// TIA Portal V17 export
// export: Created 2022-03-18T11:15:14.7636384Z, ExportSetting WithDefaults, DisplayName Totally Integrated Automation Portal, DisplayVersion V17, DisplayName TIA Portal Openness, DisplayVersion V17, DisplayName TIA Portal Version Control Interface, DisplayVersion V17, DisplayName SINAMICS Startdrive Advanced, DisplayVersion V17, DisplayName SINAMICS Startdrive G130, G150, S120, S150, SINAMICS MV, S210, DisplayVersion V17, DisplayName SINAMICS Startdrive G110M, G120, G120C, G120D, G120P, G115D, DisplayVersion V17, DisplayName STEP 7 Professional, DisplayVersion V17, DisplayName STEP 7 Safety, DisplayVersion V17, DisplayName WinCC Advanced / Unified PC, DisplayVersion V17
VAR_GLOBAL   // PLC tag table "Default tag table"
   M1_out AT %Q200.0 : "M_out";
   M1_in AT %I200.0 : "M_in";
   M2_out AT %Q219.0 : "M_out";
   M2_in AT %I209.0 : "M_in";
   M3_out AT %Q238.0 : "M_out";
   M3_in AT %I218.0 : "M_in";
   M4_out AT %Q257.0 : "M_out";
   M4_in AT %I227.0 : "M_in";
   M5_out AT %Q276.0 : "M_out";
   M5_in AT %I236.0 : "M_in";
   M6_out AT %Q295.0 : "M_out";
   M6_in AT %I245.0 : "M_in";
   M7_out AT %Q314.0 : "M_out";
   M7_in AT %I254.0 : "M_in";
   M8_out AT %Q333.0 : "M_out";
   M8_in AT %I263.0 : "M_in";
   M9_out AT %Q352.0 : "M_out";
   M9_in AT %I272.0 : "M_in";
   M10_out AT %Q371.0 : "M_out";
   M10_in AT %I281.0 : "M_in";
   M11_out AT %Q390.0 : "M_out";
   M11_in AT %I290.0 : "M_in";
   M12_out AT %Q409.0 : "M_out";
   M12_in AT %I299.0 : "M_in";
   M13_out AT %Q428.0 : "M_out";
   M13_in AT %I308.0 : "M_in";
   M14_out AT %Q447.0 : "M_out";
   M14_in AT %I317.0 : "M_in";
   M15_out AT %Q466.0 : "M_out";
   M15_in AT %I326.0 : "M_in";
   M16_out AT %Q485.0 : "M_out";
   M16_in AT %I335.0 : "M_in";
   M17_out AT %Q504.0 : "M_out";
   M17_in AT %I344.0 : "M_in";
   M18_out AT %Q523.0 : "M_out";
   M18_in AT %I353.0 : "M_in";
END_VAR
